FUNCTION_BLOCK EmergencySludgeBuffer (* CAT Function Block Type *)
  (* Standard: 61499-2 *)
  (* Version 0.0, 7/4/2026, Schneider Electric, template *)
  PACKAGE SE.Nereda;
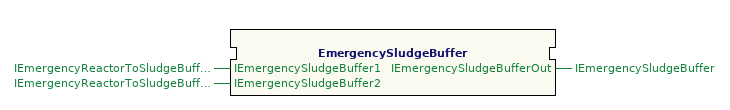
  SOCKETS
    IEmergencySludgeBuffer1 : IEmergencyReactorToSludgeBuffer;
    IEmergencySludgeBuffer2 : IEmergencyReactorToSludgeBuffer;
  END_SOCKETS
  PLUGS
    IEmergencySludgeBufferOut : IEmergencySludgeBuffer;
  END_PLUGS
  (* 01 - FUNCTIONNAL INPUT INTERFACE *)
  (* 00 - INITIALIZATION *)
  (* 05 - LOGIC *)
  (* 06 - HMI INTERFACE *)
  (* 03 - FIELD INTERFACE *)
  (* 02 - FUNCTIONNAL OUTPUT INTERFACE *)
  (* Emergency Recipe Logic *)
  (* 04 - CHILDREN *)
  (* 4A - TYPICALS *)
  (* Steps Durations *)
  FBS
    INIT : plcStart(Prio := 50, Delay := T#0ms);
    IThis : EmergencySludgeBuffer_HMI(QI := TRUE);
    Step1_Feed : E_DELAY_V_D_ZERO;
    Step2_Wait : E_DELAY_V_D_ZERO;
    Step3_SludgeDischarge : E_DELAY_V_D_ZERO;
    Step4_SupernatantDischarge : E_DELAY_V_D_ZERO;
    FeedStarted : boolValueChanged;
    EmergencyRecipeSequence : EmergencyRecipeSequenceSludgeBuffer;
    MultiReactors1 : MultiReactors;
    FB_SBL1 : COMPARE_1329C2AB45109BAAB; {SET_ATTRIBUTE(Configuration.GenericFBType.InterfaceParams, Runtime.Standard#CNT:=2;IN${CNT$}:REAL)}
    FB_SBL2 : COMPARE_1329C2AB45109BAAB; {SET_ATTRIBUTE(Configuration.GenericFBType.InterfaceParams, Runtime.Standard#CNT:=2;IN${CNT$}:REAL)}
  END_FBS
  EVENT_CONNECTIONS
    Step1_Feed.1457E63E0C241C83 TO EmergencyRecipeSequence.62A0C79B5D89C4FB;
    Step2_Wait.1457E63E0C241C83 TO EmergencyRecipeSequence.24741A0901B103DB;
    Step3_SludgeDischarge.1457E63E0C241C83 TO EmergencyRecipeSequence.FEA4481ED0C2A43C;
    Step4_SupernatantDischarge.1457E63E0C241C83 TO EmergencyRecipeSequence.9041C273A86FC2E4;
    EmergencyRecipeSequence.BFFB06EAE80CA24C TO Step1_Feed.START;
    EmergencyRecipeSequence.899C844BE45E6C4D TO Step1_Feed.STOP;
    EmergencyRecipeSequence.758107C20AA8F48B TO Step2_Wait.START;
    EmergencyRecipeSequence.18CD3557BE39D07B TO Step2_Wait.STOP;
    EmergencyRecipeSequence.77F2040F9E65C9AB TO Step3_SludgeDischarge.START;
    EmergencyRecipeSequence.728874E1FE8923C2 TO Step3_SludgeDischarge.STOP;
    EmergencyRecipeSequence.F0D24A0013391FCB TO Step4_SupernatantDischarge.START;
    EmergencyRecipeSequence.DBC21B10FAB6B6D6 TO Step4_SupernatantDischarge.STOP;
    Step1_Feed.INITO TO Step2_Wait.INIT;
    Step2_Wait.INITO TO Step3_SludgeDischarge.INIT;
    Step3_SludgeDischarge.INITO TO Step4_SupernatantDischarge.INIT;
    MultiReactors1.772BFDB0187DD8F7 TO EmergencyRecipeSequence.68E2F3B4BFF358D6;
    MultiReactors1.514B8DC5CA25B31C TO EmergencyRecipeSequence.25F0D728C2D36669;
    MultiReactors1.DB00BC0592E0C931 TO EmergencyRecipeSequence.8BD9ED85505D599F;
    MultiReactors1.DB00BC0592E0C931 TO EmergencyRecipeSequence.5327B87255632EDE;
    IEmergencySludgeBufferOut.01031D6AC20FAB24 TO EmergencyRecipeSequence.675981AE93E2378A;
    EmergencyRecipeSequence.BFFB06EAE80CA24C TO IEmergencySludgeBufferOut.37BB0210227B4D88;
    EmergencyRecipeSequence.758107C20AA8F48B TO IEmergencySludgeBufferOut.B8FB7A13CF18B1CA;
    EmergencyRecipeSequence.77F2040F9E65C9AB TO IEmergencySludgeBufferOut.7AF6A44EC4713EB1;
    EmergencyRecipeSequence.F0D24A0013391FCB TO IEmergencySludgeBufferOut.6CE3EC6EFAA8A173;
    EmergencyRecipeSequence.DBC21B10FAB6B6D6 TO IEmergencySludgeBufferOut.6CE3EC6EFAA8A173;
    EmergencyRecipeSequence.728874E1FE8923C2 TO IEmergencySludgeBufferOut.7AF6A44EC4713EB1;
    EmergencyRecipeSequence.18CD3557BE39D07B TO IEmergencySludgeBufferOut.B8FB7A13CF18B1CA;
    EmergencyRecipeSequence.899C844BE45E6C4D TO IEmergencySludgeBufferOut.37BB0210227B4D88;
    IEmergencySludgeBufferOut.BBC4AE70863ED310 TO EmergencyRecipeSequence.5F230DB7635D55AE;
    IEmergencySludgeBufferOut.FD5E09F22E2FB8C9 TO EmergencyRecipeSequence.5F230DB7635D55AE;
    IEmergencySludgeBufferOut.D7091D88C8316783 TO EmergencyRecipeSequence.5F230DB7635D55AE;
    IEmergencySludgeBufferOut.4C01A7A01C491F67 TO EmergencyRecipeSequence.5F230DB7635D55AE;
    MultiReactors1.772BFDB0187DD8F7 TO IEmergencySludgeBufferOut.4D4A6D622AA6CDB1;
    INIT.FIRST_INIT TO IThis.11B0EEC0AF1F6F5A;
    INIT.REDO_INIT TO IThis.11B0EEC0AF1F6F5A;
    IThis.69E91E9E46EEE4A5 TO IThis.9D2FDC03CB586F4F;
    EmergencyRecipeSequence.556D2F5B235B9790 TO IThis.C39B00E2AD0232CC;
    MultiReactors1.772BFDB0187DD8F7 TO IThis.C454C4B6A808EB9F;
    MultiReactors1.514B8DC5CA25B31C TO IThis.FD84EE6824F2A446;
    IThis.69E91E9E46EEE4A5 TO Step1_Feed.INIT;
    IThis.72CBF4E7BB40B16D TO IEmergencySludgeBufferOut.7AF6A44EC4713EB1;
    IThis.024A635046F06C0B TO IEmergencySludgeBufferOut.6CE3EC6EFAA8A173;
    IThis.2C6032014B484D68 TO EmergencyRecipeSequence.5D8E05AD95449444;
    IThis.99E42A5A4A27FD06 TO FB_SBL1.REQ;
    FB_SBL1.CNF TO EmergencyRecipeSequence.F6AE117EB4EE709F;
    IThis.6604743EA757FACA TO FB_SBL2.REQ;
    FB_SBL2.CNF TO EmergencyRecipeSequence.C960811A6435E9DC;
  END_CONNECTIONS
  DATA_CONNECTIONS
    Step1_Feed.716D3F3042596C89 TO EmergencyRecipeSequence.CA116731A496187E;
    Step2_Wait.716D3F3042596C89 TO EmergencyRecipeSequence.356882B50FEB9A7D;
    Step3_SludgeDischarge.716D3F3042596C89 TO EmergencyRecipeSequence.111361C8BEDF440B;
    Step4_SupernatantDischarge.716D3F3042596C89 TO EmergencyRecipeSequence.82CEB92F735FC5D4;
    MultiReactors1.11DE90CF81B60953 TO EmergencyRecipeSequence.C537A25E1616B854;
    MultiReactors1.BE19DC348C3D36F1 TO EmergencyRecipeSequence.53ADC5A2738A60DC;
    MultiReactors1.90CEC3EB9AF77987 TO EmergencyRecipeSequence.EB24B639967D6395;
    MultiReactors1.E181861A95CF66B5 TO EmergencyRecipeSequence.A1908D16CCF1B616;
    MultiReactors1.9EA7F0E93CE8C3C8 TO EmergencyRecipeSequence.E5E1D6F5F3F937A2;
    IEmergencySludgeBufferOut.91843A91DDCD538F TO EmergencyRecipeSequence.6882FED931B8B218;
    EmergencyRecipeSequence.8B42F21C51560908 TO IEmergencySludgeBufferOut.0CCCE0E6A38C4CC4;
    EmergencyRecipeSequence.A9E8FE003DEE6E89 TO IEmergencySludgeBufferOut.2D97C7DF176F1821;
    EmergencyRecipeSequence.2A15B42D80F87BCA TO IEmergencySludgeBufferOut.CC5E48971A6D3B85;
    EmergencyRecipeSequence.A11B93FCF2C8455F TO IEmergencySludgeBufferOut.FDC6C047971AF4AB;
    IEmergencySludgeBufferOut.D440A766CB8B17CF TO EmergencyRecipeSequence.02C5FE17473E63ED;
    IEmergencySludgeBufferOut.862A2E6EE70C20AF TO EmergencyRecipeSequence.5FBA38ABF9198C98;
    IEmergencySludgeBufferOut.695399F703F77E2B TO EmergencyRecipeSequence.69F1D0FE13048380;
    IEmergencySludgeBufferOut.76FC2A554E83498F TO EmergencyRecipeSequence.9F29B8C1612DCC07;
    MultiReactors1.11DE90CF81B60953 TO IEmergencySludgeBufferOut.A1711B52790021B0;
    EmergencyRecipeSequence.1A64065878672AC0 TO IThis.B3535F417A0074C5;
    MultiReactors1.11DE90CF81B60953 TO IThis.71DB4288F980DD7A;
    MultiReactors1.BE19DC348C3D36F1 TO IThis.7498551BC2E13233;
    IThis.D3644ED70524C0F1 TO Step1_Feed.DT1;
    IThis.33D4356E329ECCF2 TO Step2_Wait.DT1;
    IThis.9B01CEED6ECAE668 TO Step3_SludgeDischarge.DT1;
    IThis.11E3ABF20E7068A4 TO Step4_SupernatantDischarge.DT1;
    IThis.109297249ED70180 TO IEmergencySludgeBufferOut.290CB544BD4AF7E0;
    IThis.14CC246E4360C5FD TO IEmergencySludgeBufferOut.D5F6310F45243454;
    IThis.7C70A0C13C0753EB TO EmergencyRecipeSequence.BEC170C6FAF98287;
    IEmergencySludgeBufferOut.91843A91DDCD538F TO FB_SBL1.IN1;
    IThis.345A6464C12A0050 TO FB_SBL1.IN2;
    FB_SBL1.LE TO EmergencyRecipeSequence.7A1CAB8AE52AE374;
    IEmergencySludgeBufferOut.91843A91DDCD538F TO FB_SBL2.IN1;
    IThis.BEDB1A4BAB5FF8C7 TO FB_SBL2.IN2;
    FB_SBL2.LE TO EmergencyRecipeSequence.CB5D14E9C5586FB9;
  END_CONNECTIONS
  ADAPTER_CONNECTIONS
    IEmergencySludgeBuffer1 TO MultiReactors1.6D0E314F030D4C27;
    IEmergencySludgeBuffer2 TO MultiReactors1.77861C060F39F3A3;
  END_CONNECTIONS
END_FUNCTION_BLOCK
